// SIMATIC S7-200 project (STEP 7-Micro/WIN), CPU 224XP REL 02.01

ORGANIZATION_BLOCK 主程序:OB1
TITLE=程序注释
BEGIN
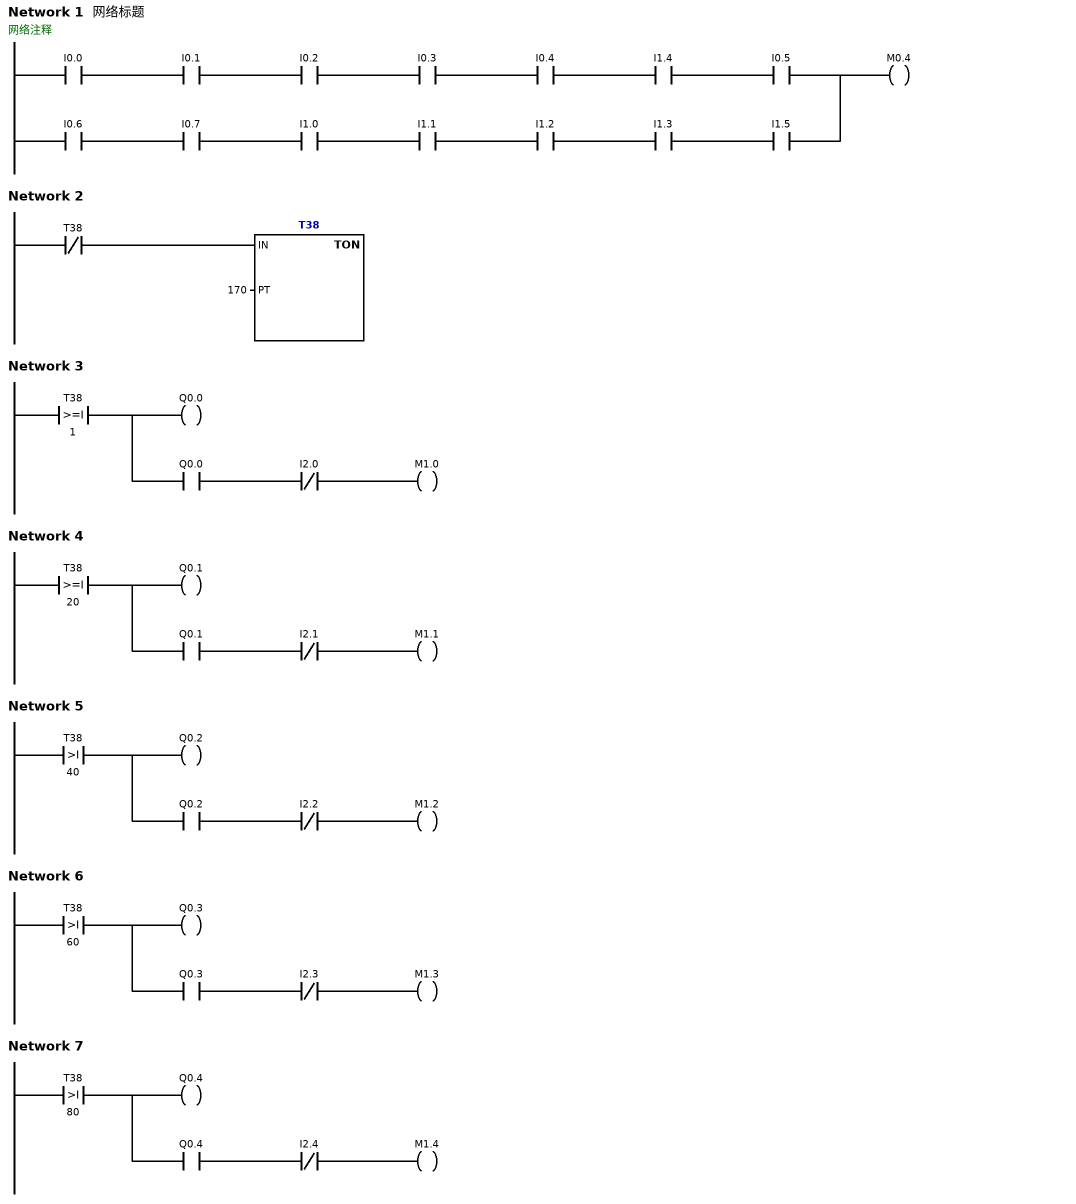
Network 1 // 网络标题
// 网络注释
LD     I0.0
A      I0.1
A      I0.2
A      I0.3
A      I0.4
A      I1.4
A      I0.5
LD     I0.6
A      I0.7
A      I1.0
A      I1.1
A      I1.2
A      I1.3
A      I1.5
OLD
=      M0.4
Network 2
LDN    T38
TON    T38, 170
Network 3
LDW>=  T38, 1
=      Q0.0
A      Q0.0
AN     I2.0
=      M1.0
Network 4
LDW>=  T38, 20
=      Q0.1
A      Q0.1
AN     I2.1
=      M1.1
Network 5
LDW>   T38, 40
=      Q0.2
A      Q0.2
AN     I2.2
=      M1.2
Network 6
LDW>   T38, 60
=      Q0.3
A      Q0.3
AN     I2.3
=      M1.3
Network 7
LDW>   T38, 80
=      Q0.4
A      Q0.4
AN     I2.4
=      M1.4
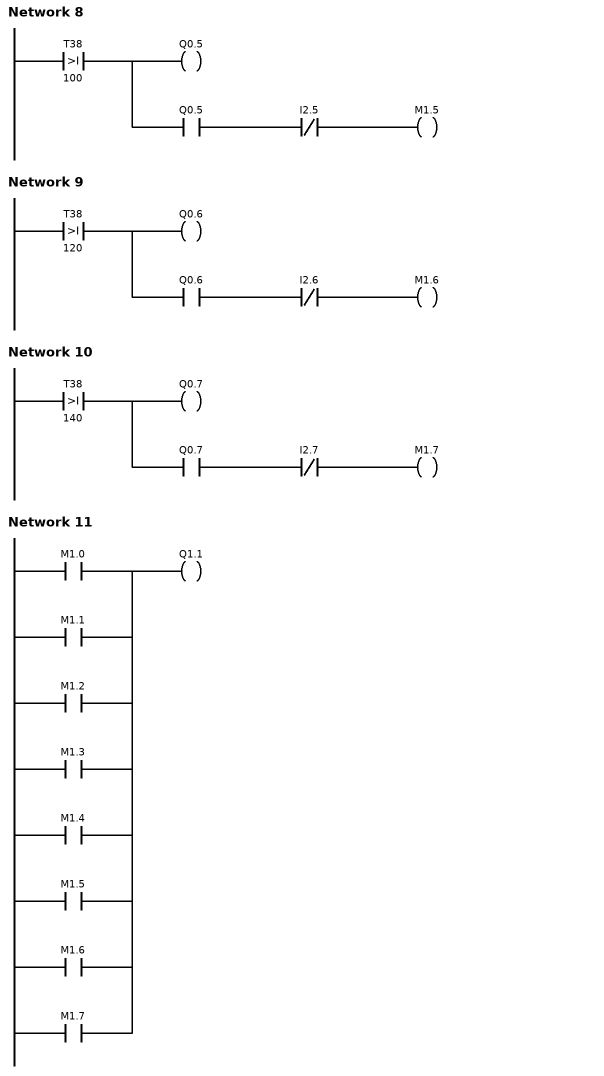
Network 8
LDW>   T38, 100
=      Q0.5
A      Q0.5
AN     I2.5
=      M1.5
Network 9
LDW>   T38, 120
=      Q0.6
A      Q0.6
AN     I2.6
=      M1.6
Network 10
LDW>   T38, 140
=      Q0.7
A      Q0.7
AN     I2.7
=      M1.7
Network 11
LD     M1.0
O      M1.1
O      M1.2
O      M1.3
O      M1.4
O      M1.5
O      M1.6
O      M1.7
=      Q1.1
END_ORGANIZATION_BLOCK
